howbig := sizeof(ptArray^);
// Clear error bit
q_xError := FALSE;
IF iMessageLen = iCurrIndex THEN
    //Dont do a damn thing
    ;
// Check the remaining length and shift amount summed is not greater than the total array width.
ELSIF iSize < (iMessageLen - iCurrIndex) + iShift THEN
    q_xError := TRUE;
ELSE// MEMMOVE from 1+ the current index to the remaining length by the shift amount
    IF MEMMOVE(srcAddr:=(ptArray + iCurrIndex + 1), destAddr:=(ptArray + iCurrIndex + 1 + iShift), n:=INT_TO_UDINT(iMessageLen + 1 - iCurrIndex)) =0 THEN
        q_xError := TRUE;
    END_IF
END_IF

END_FUNCTION_BLOCK

// ---- POUs/Sensirion/fSHDLCChecksum.TcPOU
FUNCTION fSHDLCChecksum : BYTE
VAR_INPUT
    i_bAdr	:	BYTE;
    i_bCmd	:	BYTE;
    i_bLen	:	BYTE;
    i_pbaTxData	:	POINTER TO BYTE;
END_VAR
VAR
    iIndex	:	INT;
END_VAR

(* Checksum is calc like so
Sum all the bytes within the frame
Take the LSN ie. nibble of the result and invert it
*)

fSHDLCChecksum := i_bAdr + i_bCmd + i_bLen;

IF i_bLen > 0 THEN
FOR iIndex:=0 TO BYTE_TO_INT(i_bLen)DO
    fSHDLCChecksum := fSHDLCChecksum + i_pbaTxData^;
    i_pbaTxData := i_pbaTxData + 1;
END_FOR
END_IF

// Inverting LSN
fSHDLCChecksum := fSHDLCChecksum XOR 16#FF;

END_FUNCTION

// ---- POUs/PCM/FB_PressureControlModule.TcPOU
// Encapsulation of a pressure control module.
// A. Wallace, 2019-10-22
// Support for 2 proportionairs, 4 generic analog inputs (usually a pressure gauge
// and two shimadzu ports.
FUNCTION_BLOCK FB_PressureControlModule
VAR_INPUT
END_VAR
VAR_OUTPUT
END_VAR
VAR_IN_OUT
END_VAR
VAR
    {attribute 'pytmc' := '
        pv: IO
     '}
    stBaseIO : ST_M3DeviceBaseIO;

    stSerial1 : ST_SerialComm;
    stSerial2 : ST_SerialComm;

    fbSerial1 : FB_SerialCommWrapper;
    fbSerial2 : FB_SerialCommWrapper;

    {attribute 'pytmc' := '
        pv: PropAir:01
     '}
    stPropAir1 : ST_Proportionair;
    {attribute 'pytmc' := '
        pv: PropAir:02
     '}
    stPropAir2 : ST_Proportionair;

    PropAir1 : FB_ProportionairRegulator;
    PropAir2 : FB_ProportionairRegulator;
END_VAR

PropAir1(iq_stRegProp:=stPropAir1);
PropAir2(iq_stRegProp:=stPropAir2);

ACTION SerialComm:
fbSerial1(stSerialComm := stSerial1);
fbSerial2(stSerialComm := stSerial2);
END_ACTION

END_FUNCTION_BLOCK

// ---- POUs/Regulators/FB_ProportionairRegulator.TcPOU
FUNCTION_BLOCK FB_ProportionairRegulator
VAR_INPUT
END_VAR
VAR_OUTPUT
END_VAR
VAR_IN_OUT
    iq_stRegProp	:	ST_Proportionair;
END_VAR
VAR

END_VAR

(* A. Wallace 2015-10-7
Proportionair regulator control *)

(* Pressure signal conversion, max pressure out 1000 (I think...) *)
iq_stRegProp.iPressure := REAL_TO_INT(1000 * (MAX(0,INT_TO_REAL(iq_stRegProp.i_iPressRB)) / 32767));

iq_stRegProp.iSetpoint := LIMIT(iq_stRegProp.iLoLimit, iq_stRegProp.iSetpoint, iq_stRegProp.iHiLimit);

iq_stRegProp.q_iPressCt := REAL_TO_INT( (INT_TO_REAL(iq_stRegProp.iSetpoint)/1000)*32767);

END_FUNCTION_BLOCK

// ---- POUs/GasManifold/FB_GasManifold.TcPOU
FUNCTION_BLOCK FB_GasManifold
VAR_INPUT
END_VAR
VAR_OUTPUT
END_VAR
VAR
    {attribute 'pytmc' := '
        pv: IO
     '}
    stBaseIO : ST_M3DeviceBaseIO;


    {attribute 'pytmc' := '
        pv: Valve
     '}
    stValve : ARRAY [1..MANIFOLD_VALVES] OF ST_ManifoldValve;
    fbValve : ARRAY [1..MANIFOLD_VALVES] OF FB_ManiValve;
    idx : int;
END_VAR
VAR CONSTANT
    MANIFOLD_VALVES : INT := 7;
END_VAR

FOR idx := 1 to MANIFOLD_VALVES DO
    stValve[idx].xILK := TRUE; // these valves have no interlock
    fbValve[idx](iq_valve := stValve[idx]);
END_FOR

END_FUNCTION_BLOCK

// ---- POUs/GasManifold/FB_ManiValve.TcPOU
FUNCTION_BLOCK FB_ManiValve
VAR_INPUT
END_VAR
VAR_OUTPUT
END_VAR
VAR_IN_OUT
    iq_valve	:	ST_ManifoldValve;
END_VAR
VAR
END_VAR

(* Basic valve control block *)
IF NOT iq_valve.xILK THEN
    iq_valve.xSW := FALSE;
END_IF

iq_valve.qxDO := NOT (iq_valve.xILK and iq_valve.xSW); // These are normally open valves, qxDO closes the valve

END_FUNCTION_BLOCK

// ---- POUs/Bronkhorst/FB_BronkhorstMFM.TcPOU
FUNCTION_BLOCK FB_BronkhorstMFM
VAR_INPUT
END_VAR
VAR_OUTPUT
END_VAR
VAR
        {attribute 'pytmc' := '
            pv:
         '}
        stMFM	:	ST_BhElFlow;
END_VAR

END_FUNCTION_BLOCK

// ---- POUs/DigitalOutput/FB_SolenoidPair.TcPOU
FUNCTION_BLOCK FB_SolenoidPair
VAR_INPUT
END_VAR
VAR_OUTPUT
END_VAR
VAR_IN_OUT
END_VAR
VAR
    {attribute 'pytmc' := '
        pv: Valve:01:Open
        io: io
     '}
    q_xDO1 AT %Q*	:	BOOL;
    {attribute 'pytmc' := '
        pv: Valve:02:Open
        io: io
     '}
    q_xDO2 AT %Q*	:	BOOL;

    {attribute 'pytmc' := '
        pv: Switch
        io: o
     '}
    i_xEpics AT %I* : BOOL; // open A when False, open B when True

    {attribute 'pytmc' := '
        pv: Debug
        io: o
     '}
    i_xDebug AT %I* : BOOL; // if True, do not set valves according to i_xEpics
END_VAR

(* If debug, set independently. Else, only open one valve according to i_xEpics *)
IF NOT i_xDebug THEN
    q_xDO1 := NOT i_xEpics;
    q_xDO2 := i_xEpics;
END_IF

END_FUNCTION_BLOCK

// ---- POUs/Helpers/FB_EcatDiag.TcPOU
FUNCTION_BLOCK FB_EcatDiag
VAR_INPUT
    i_AMSNetId	:	AMSNETID; //Connect this to an AMSNETID structure as a PLC input. Then link the input to the AMSNETID name in the master info.
    i_xFirstPass	:	BOOL;
END_VAR
VAR_OUTPUT
    q_xAllStatesGood	:	BOOL;
END_VAR
VAR
    sNetId : T_AmsNetId;
    astTermStates : ARRAY[1..256] OF ST_EcSlaveState;

    fbGetAllSlaveStates     : FB_EcGetAllSlaveStates;
    ftReset	: F_TRIG;

    iterator: INT;
END_VAR

//Create the net ID string
sNetID := F_CreateAmsNetId(i_AMSNetId);

//Query the state of all terminals, collect in astTermStates
ftReset(CLK:=fbGetAllSlaveStates.bBusy OR i_xFirstPass);
fbGetAllSlaveStates.bExecute := ftReset.Q;
fbGetAllSlaveStates(sNetId:=sNetId, pStateBuf := ADR(astTermStates), cbBufLen:=SIZEOF(astTermStates));
//Keep checking...

//Cycle through each entry in the array and check if we have anyone not in OP and that the link state is good.
// If so, then set our global IO bad boolean.
IF fbGetAllSlaveStates.nSlaves > 0 THEN
    q_xAllStatesGood := TRUE;
FOR iterator := 1 TO (fbGetAllSlaveStates.nSlaves -1) BY 1
    DO
    IF NOT( (astTermStates[iterator].deviceState = EC_DEVICE_STATE_OP) AND (astTermStates[iterator].linkState = EC_LINK_STATE_OK)) THEN
        q_xAllStatesGood := FALSE;
    END_IF
END_FOR
END_IF

END_FUNCTION_BLOCK

// ---- POUs/p_ALI.TcPOU
PROGRAM p_ALI
VAR
    fbALI_A	:	FB_ALI;
END_VAR

fbALI_A(iq_Injector:=stALI);

END_PROGRAM

// ---- POUs/p_Autosave.TcPOU
PROGRAM p_Autosave
VAR
END_VAR

(* If first pass, copy all persistent variables (which should be intialized to old values) back into the operational variables *)
IF g_xFirstPass THEN

    stRegProp1 := gp_stRegProp1;
    stRegProp2 := gp_stRegProp2;
    stRegProp3 := gp_stRegProp3;
    stRegProp4 := gp_stRegProp4;

ELSE
    gp_stRegProp1 := stRegProp1;
    gp_stRegProp2 := stRegProp2;
    gp_stRegProp3 := stRegProp3;
    gp_stRegProp4 := stRegProp4;

END_IF

END_PROGRAM

// ---- POUs/p_AutoWash.TcPOU
PROGRAM p_AutoWash
VAR



END_VAR

END_PROGRAM

// ---- POUs/p_CoolerShaker.TcPOU
PROGRAM p_CoolerShaker
VAR

afbTECDriver	:	ARRAY[1..3] OF FB_TECDriver;

    index: INT :=1 ;
END_VAR


stTECCtrl[1].sAddress := '01'; //62 is 98 in hex which is default address
stTECCtrl[2].sAddress := '02';
stTECCtrl[3].sAddress := '62';

stTECCtrl[1].diTempSetpoint := 30; //98 in hex which is default address
stTECCtrl[2].diTempSetpoint := 30;
stTECCtrl[3].diTempSetpoint := 30;

afbTECDriver[index](
    i_xExecute:= TRUE,
    i_tTimeOut:= t#1s,
    i_stControl:= stTECCtrl[index],
    iq_stSerialRXBuffer:= SerialRXBuffer_CoolerShakerTEC,
    iq_stSerialTXBuffer:= SerialTXBuffer_CoolerShakerTEC,
    q_stStatus=>stTECStatus[index]);

IF afbTECDriver[index].q_xDone OR
    afbTECDriver[index].q_xError OR
    afbTECDriver[index].q_xTimeout THEN
    (* reset function for next time *)
    afbTECDriver[index](i_xExecute:=FALSE, iq_stSerialRXBuffer:= SerialRXBuffer_CoolerShakerTEC, iq_stSerialTXBuffer:=  SerialTXBuffer_CoolerShakerTEC);

    index := index + 1;
    IF index > 2 THEN index := 1; END_IF

END_IF

END_PROGRAM

// ---- POUs/TEC/FB_TECDriver.TcPOU
FUNCTION_BLOCK FB_TECDriver

VAR_INPUT
    i_xExecute				: BOOL;					(* rising edge execute *)
    i_tTimeOut				: TIME := t#10s;  		(* Maximum wait time for reply *)
    i_stControl				: ST_TECControl;
END_VAR
VAR_OUTPUT
    q_xDone					: BOOL;
    q_xError				: BOOL;
    q_xWarning				: BOOL;					(* set in the event of an unexpected reply *)
    q_xTimeout				: BOOL;
    q_sResult				: STRING(255);
    q_sLastSentString		: ARRAY[1..40] OF STRING;				(* Last String Sent to Serial Device - for debugging *)
    q_sLastReceivedString	: ARRAY[1..40] OF STRING;				(* Last String Received from Serial Device - for debugging *)
    q_stStatus				: ST_TECStatus;
END_VAR
VAR_IN_OUT
    iq_stSerialRXBuffer 	: ComBuffer;
    iq_stSerialTXBuffer 	: ComBuffer;
END_VAR
VAR
    rtExecute				: R_TRIG;
    iStep					: INT;
    sSendData				: STRING;
    fbTECTransaction		: FB_TECTransaction;
    (*fbFormatString			: FB_FormatString;*)
    (*fbSplit					: FB_Split255;*)
    asReplyFields			: ARRAY[1..20] OF T_MaxString;
    wChecksum: WORD;
    rtStartIntegration: R_TRIG;
    rtEndReset: R_TRIG;

    sWorking: STRING;
    strResponseExpected: STRING;
    diWorking	:	DINT;
END_VAR

(* This function block performs serial communication with a TC-36-25 TEC Driver *)

(* rising edge trigger *)
rtExecute(CLK:= i_xExecute);
IF rtExecute.Q  THEN
    q_xDone	:= FALSE;
    q_xError := FALSE;
    q_xWarning := FALSE;
    q_xTimeout := FALSE;
    q_sResult:= '';
    fbTECTransaction( i_xExecute:= FALSE, iq_stSerialRXBuffer:= iq_stSerialRXBuffer, iq_stSerialTXBuffer:= iq_stSerialTXBuffer );  (* reset *)

    iStep := 10;
END_IF

CASE iStep OF
    0: (* idle *)
        ;

    10: (* Get Current Temperature *)
        fbTECTransaction(
            i_xExecute:= TRUE,
            i_sAddress:=i_stControl.sAddress,
            i_sCmd:= '01',
            i_diParameter := 0,
            i_tTimeOut:= i_tTimeOut,
            iq_stSerialRXBuffer:= iq_stSerialRXBuffer,
            iq_stSerialTXBuffer:= iq_stSerialTXBuffer,
            i_CmdFlag :=FALSE);

        IF fbTECTransaction.q_xError THEN
            q_sResult := CONCAT('in Step 10 serial transaction failed with message: ', fbTECTransaction.q_sResult);
            iStep := 9000;
        ELSIF fbTECTransaction.q_xDone THEN
            q_stStatus.sReply := fbTECTransaction.q_sResponseData;
            sWorking :=LEFT(q_stStatus.sReply, 8);
            sWorking := CONCAT('16#', sWorking);
            q_stStatus.diTemp1 := STRING_TO_DINT(sWorking);
            fbTECTransaction( i_xExecute:= FALSE, iq_stSerialRXBuffer:= iq_stSerialRXBuffer, iq_stSerialTXBuffer:= iq_stSerialTXBuffer, i_CmdFlag :=FALSE);  (* reset *)
            iStep := 20;

        END_IF
    20: (* Read setpoint *)
        fbTECTransaction(
            i_xExecute:= TRUE,
            i_sAddress:=i_stControl.sAddress,
            i_sCmd:= '03', // command
            i_diParameter := 0, // always zero for query
            i_tTimeOut:= i_tTimeOut,
            iq_stSerialRXBuffer:= iq_stSerialRXBuffer,
            iq_stSerialTXBuffer:= iq_stSerialTXBuffer,
            i_CmdFlag :=FALSE);

        IF fbTECTransaction.q_xError THEN
            q_sResult := CONCAT('in Step 20 serial transaction failed with message: ', fbTECTransaction.q_sResult);
            iStep := 9000;
        ELSIF fbTECTransaction.q_xDone THEN
            q_stStatus.sReply := fbTECTransaction.q_sResponseData;
            sWorking :=LEFT(q_stStatus.sReply, 8);
            sWorking := CONCAT('16#', sWorking);
            q_stStatus.diSetPoint := STRING_TO_DINT(sWorking);
            fbTECTransaction( i_xExecute:= FALSE, iq_stSerialRXBuffer:= iq_stSerialRXBuffer, iq_stSerialTXBuffer:= iq_stSerialTXBuffer, i_CmdFlag :=FALSE);  (* reset *)
            iStep := 25;
        END_IF

    25: (* Read output ON/OFF *)
        fbTECTransaction(
            i_xExecute:= TRUE,
            i_sAddress:=i_stControl.sAddress,
            i_sCmd:= '46', // command
            i_diParameter := 0, // always zero for query
            i_tTimeOut:= i_tTimeOut,
            iq_stSerialRXBuffer:= iq_stSerialRXBuffer,
            iq_stSerialTXBuffer:= iq_stSerialTXBuffer,
            i_CmdFlag :=FALSE);

        IF fbTECTransaction.q_xError THEN
            q_sResult := CONCAT('in Step 25 serial transaction failed with message: ', fbTECTransaction.q_sResult);
            iStep := 9000;
        ELSIF fbTECTransaction.q_xDone THEN
            q_stStatus.sReply := fbTECTransaction.q_sResponseData;
            sWorking :=LEFT(q_stStatus.sReply, 8);
            sWorking := CONCAT('16#', sWorking);
            diWorking := STRING_TO_DINT(sWorking);
            q_stStatus.xOutputOn := DINT_TO_BOOL(diWorking);
            A_ResetTransaction();
            iStep := 30;
        END_IF

    30: (* Read the alarm status *)
        fbTECTransaction(
            i_xExecute:= TRUE,
            i_sAddress:=i_stControl.sAddress,
            i_sCmd:= '05', // command
            i_diParameter := 0, // always zero for query
            i_tTimeOut:= i_tTimeOut,
            iq_stSerialRXBuffer:= iq_stSerialRXBuffer,
            iq_stSerialTXBuffer:= iq_stSerialTXBuffer,
            i_CmdFlag :=FALSE);

        IF fbTECTransaction.q_xError THEN
            q_sResult := CONCAT('in Step 10 serial transaction failed with message: ', fbTECTransaction.q_sResult);
            iStep := 9000;
        ELSIF fbTECTransaction.q_xDone THEN
            q_stStatus.sReply := fbTECTransaction.q_sResponseData;
            sWorking :=LEFT(q_stStatus.sReply, 8);
            sWorking := CONCAT('16#', sWorking);
            diWorking := STRING_TO_DINT(sWorking);

            //Alarm assignment
            q_stStatus.xHiTemp	:=	diWorking.0;
            q_stStatus.xLoTemp	:=	diWorking.1;
            q_stStatus.xLoTemp	:=	diWorking.2;
            q_stStatus.xOverCurrent	:=	diWorking.3;
            q_stStatus.xOpenInput1	:=	diWorking.4;
            q_stStatus.xOpenInput2	:=	diWorking.5;
            q_stStatus.xDriverLowVoltage	:=	diWorking.6;

            fbTECTransaction( i_xExecute:= FALSE, iq_stSerialRXBuffer:= iq_stSerialRXBuffer, iq_stSerialTXBuffer:= iq_stSerialTXBuffer, i_CmdFlag :=FALSE);  (* reset *)
            iStep := 40;
        END_IF

    40: (* Output Power *)
        fbTECTransaction(
            i_xExecute:= TRUE,
            i_sAddress:=i_stControl.sAddress,
            i_sCmd:= '02', // command
            i_diParameter := 0, // always zero for query
            i_tTimeOut:= i_tTimeOut,
            iq_stSerialRXBuffer:= iq_stSerialRXBuffer,
            iq_stSerialTXBuffer:= iq_stSerialTXBuffer,
            i_CmdFlag :=FALSE);

        IF fbTECTransaction.q_xError THEN
            q_sResult := CONCAT('in Step 10 serial transaction failed with message: ', fbTECTransaction.q_sResult);
            iStep := 9000;
        ELSIF fbTECTransaction.q_xDone THEN
            q_stStatus.sReply := fbTECTransaction.q_sResponseData;
            sWorking :=LEFT(q_stStatus.sReply, 8);
            sWorking := CONCAT('16#', sWorking);
            diWorking := STRING_TO_DINT(sWorking);

            q_stStatus.diPercentOut := (diWorking/511)*100; //in percentage

            fbTECTransaction( i_xExecute:= FALSE, iq_stSerialRXBuffer:= iq_stSerialRXBuffer, iq_stSerialTXBuffer:= iq_stSerialTXBuffer, i_CmdFlag :=FALSE);  (* reset *)
            iStep := 5000;
        END_IF

    5000: (* Change Setpoint *)
        IF q_stStatus.diSetpoint <> i_stControl.diTempSetpoint THEN

            fbTECTransaction(
                i_xExecute:= TRUE,
                i_sAddress:=i_stControl.sAddress,
                i_sCmd:= '1c', // command
                i_diParameter := i_stControl.diTempSetpoint,
                i_tTimeOut:= i_tTimeOut,
                iq_stSerialRXBuffer:= iq_stSerialRXBuffer,
                iq_stSerialTXBuffer:= iq_stSerialTXBuffer,
                i_CmdFlag :=TRUE);
            IF fbTECTransaction.q_xError THEN
                q_sResult := CONCAT('in Step 5000 serial transaction failed with message: ', fbTECTransaction.q_sResult);
                iStep := 9000;
            ELSIF fbTECTransaction.q_xDone THEN
                fbTECTransaction(
                     i_xExecute:= FALSE,
                    iq_stSerialRXBuffer:= iq_stSerialRXBuffer,
                    iq_stSerialTXBuffer:= iq_stSerialTXBuffer,
                    i_CmdFlag:=FALSE );  (* reset *)
                iStep := 5010;
            END_IF
        ELSE
            iStep := 5010;
        END_IF

    5010: (* Output ON/OFF *)
        IF q_stStatus.xOutputOn <> i_stControl.xOutputOn THEN

            fbTECTransaction(
                i_xExecute:= TRUE,
                i_sAddress:=i_stControl.sAddress,
                i_sCmd:= '2d', // command
                i_diParameter := BOOL_TO_DINT(i_stControl.xOutputOn),
                i_tTimeOut:= i_tTimeOut,
                iq_stSerialRXBuffer:= iq_stSerialRXBuffer,
                iq_stSerialTXBuffer:= iq_stSerialTXBuffer,
                i_CmdFlag :=TRUE);
            IF fbTECTransaction.q_xError THEN
                q_sResult := CONCAT('in Step 5010 serial transaction failed with message: ', fbTECTransaction.q_sResult);
                iStep := 9000;
            ELSIF fbTECTransaction.q_xDone THEN
                fbTECTransaction(
                     i_xExecute:= FALSE,
                    iq_stSerialRXBuffer:= iq_stSerialRXBuffer,
                    iq_stSerialTXBuffer:= iq_stSerialTXBuffer,
                    i_CmdFlag:=FALSE );  (* reset *)
                iStep := 8000;
            END_IF
        ELSE
            iStep := 8000;
        END_IF


    8000: (* done *)
        q_xDone := TRUE;
        IF q_sResult = '' THEN
            q_sResult := 'Success';
            q_stStatus.xStatusValid := TRUE;
        END_IF
        IF  i_xExecute = FALSE THEN
            q_xDone:= FALSE;
            iStep := 0;
        END_IF

    9000:
        _A_ClearStatus();
        q_xTimeout := fbTECTransaction.q_xTimeout;
        q_xError := TRUE;
        q_stStatus.xStatusValid := FALSE;


END_CASE

q_sLastSentString := fbTECTransaction.q_sLastSentString;
q_sLastReceivedString := fbTECTransaction.q_sLastReceivedString;

ACTION A_ResetTransaction:
fbTECTransaction( i_xExecute:= FALSE, iq_stSerialRXBuffer:= iq_stSerialRXBuffer, iq_stSerialTXBuffer:= iq_stSerialTXBuffer, i_CmdFlag :=FALSE);  (* reset *)
END_ACTION

ACTION _A_ClearStatus:
q_stStatus.sReply := '';
END_ACTION

END_FUNCTION_BLOCK

// ---- POUs/TEC/FB_TECTransaction.TcPOU
FUNCTION_BLOCK FB_TECTransaction
VAR_INPUT
    i_xExecute				: 	BOOL;				(* Rising edge execute *)
    i_sCmd					: 	STRING(2); 			(* Send Data *)
    i_sAddress				:	STRING(2);
    i_diParameter			:	DINT;
    i_tTimeOut				:	TIME := T#10S;  	(* Maximum wait time for reply *)
    i_CmdFlag: BOOL := FALSE;
END_VAR
VAR_OUTPUT
    q_xDone					: BOOL;
    q_sResponseData			: STRING;
    q_xError				: BOOL;
    q_xTimeout				: BOOL;
    q_sResult				: STRING;
    q_sLastSentString		: ARRAY[1..40] OF STRING;			(* Last String Sent to Serial Device - for debugging *)
    q_sLastReceivedString	: ARRAY[1..40] OF STRING;			(* Last String Received from Serial Device - for debugging *)
END_VAR
VAR_IN_OUT
    iq_stSerialRXBuffer 	: ComBuffer;
    iq_stSerialTXBuffer 	: ComBuffer;
END_VAR
VAR
    rtExecute				: R_TRIG;
    iStep					: INT;
    fbClearComBuffer		: ClearComBuffer;
    fbSendString			: SendString;
    fbReceiveString			: ReceiveString;
    sReceivedString			: STRING;
    tonTimeout				: TON;
    sSendString: STRING;
    iStringTx: INT := 1;
    iStringRx: INT := 1;

    iStringTxRx: INT := 1;
    sTxRxString: ARRAY[1..40] OF STRING;

    fbFormatParamString	:	FB_FormatString;
    fbFormatParamZPadString	:	FB_FormatString;
    fbFormatCSString	:	FB_FormatString;
    sParameter: STRING;
    iIndexChkSum: INT;
    wCsSum: WORD;
    udiParameter: UDINT;

END_VAR

(* This function block performs serial transactions with a TC-36-25 TEC Driver  *)

(* rising edge trigger *)
rtExecute(CLK:= i_xExecute);
IF rtExecute.Q THEN
    q_xDone	:= FALSE;
    q_sResponseData := '';
    q_xError := FALSE;
    q_xTimeout := FALSE;
    q_sResult:= '';
    q_sLastSentString[iStringTx] := '';
    q_sLastReceivedString[iStringRx]:= '';
    iStep := 10;
END_IF

CASE iStep OF
    0:
        ; (* idle *)

    10: (* clear com buffers *)
        fbClearComBuffer(Buffer:= iq_stSerialRXBuffer);
        fbClearComBuffer(Buffer:= iq_stSerialTXBuffer);
        (* Reset receive *)
        fbReceiveString(
            Reset:= TRUE,
            ReceivedString:= sReceivedString,
            RXbuffer:= iq_stSerialRXBuffer );
        (* build the string *)
        sSendString := CONCAT(i_sAddress, i_sCmd); (* adding the address and command/query *)
        IF i_CmdFlag THEN
            (* Convert the parameter into an 8-wide hex string twos complemented*)
            udiParameter := DINT_TO_UDINT(i_diParameter);
            fbFormatParamString(sFormat:= '%x', arg1:=F_UDINT(udiParameter)); // first convert to a string
            fbFormatParamZPadString(sFormat:='%08s', arg1:=F_STRING(fbFormatParamString.sOut));// then zero pad, because FB_Format string does not zero-pad hex strings naturally
            sParameter := fbFormatParamZPadString.sOut;
        ELSE
            sParameter := '00000000'; (* send zeros if we're querying *)
        END_IF
        (* Add parameter *)
        sSendString := CONCAT(sSendString, sParameter);

        (* Compute checksum *)
        A_Checksum();

        (* add stx at start *)
        sSendString := CONCAT('*', sSendString);
        (* append checksum *)
        fbFormatCSString(sFormat := '%02x', arg1:=F_WORD(wCsSum));
        sSendString	:= CONCAT(sSendString, fbFormatCSString.sOut);
         (*adding tail *)
        sSendString := CONCAT(sSendString,'$R'); (* add <cr> *)

        IF fbFormatParamString.bError OR fbFormatCSString.bError THEN
            q_sResult := CONCAT('In step 10 fbFormatString resulted in error: ', UDINT_TO_STRING(fbFormatParamString.nErrId));
            iStep := 9000;
        ELSE
            fbSendString( SendString:= sSendString, TXbuffer:= iq_stSerialTXBuffer );
        END_IF
        q_sLastSentString[iStringTx] := sSendString;
        IF iStringTx = 40 THEN iStringTx := 1; ELSE iStringTx := iStringTx +1; END_IF
        iStep := iStep + 10;

    20: (* Finish sending the String *)
        IF fbSendString.Busy THEN
            fbSendString( SendString:= sSendString, TXbuffer:= iq_stSerialTXBuffer );
        ELSIF fbSendString.Error <> 0 THEN
            q_sResult := CONCAT('In step 20 fbSendString resulted in error: ', INT_TO_STRING(fbSendString.Error));
            iStep := 9000;
        ELSIF NOT fbSendString.Busy THEN
            iStep:=iStep + 10;
        END_IF
        tonTimeout(IN:= FALSE);

    30: (* Get reply *)
        fbReceiveString(
            Prefix:= '*',
            Suffix:= '^',
            Timeout:= i_tTimeOut,
            Reset:= FALSE,
            ReceivedString:= sReceivedString,
            RXbuffer:= iq_stSerialRXBuffer );
        tonTimeout(IN:= TRUE, PT:= i_tTimeOut);
        IF fbReceiveString.Error <> 0 THEN
            q_sResult := CONCAT('In step 30 fbReceiveString resulted in error: ', INT_TO_STRING(fbReceiveString.Error));
            iStep := 9000;
        ELSIF fbReceiveString.RxTimeout OR tonTimeout.Q THEN
            q_sResult := 'Serial device failed to reply within timeout period';
            q_xTimeout := TRUE;
            iStep := 9000;
        ELSIF fbReceiveString.StringReceived THEN
            q_sLastReceivedString[iStringRx] := sReceivedString;
            IF iStringRx = 40 THEN iStringRx := 1; ELSE iStringRx := iStringRx +1; END_IF
            IF LEN(sReceivedString) < 2 THEN
                q_sResult := 'Reply too short.';
                iStep := 9000;
            ELSE
                (* Removing stx and ack *)
                q_sResponseData := LEFT(sReceivedString,LEN(sReceivedString)-1);
                q_sResponseData := RIGHT(q_sResponseData,LEN(q_sResponseData)-1);
                (* Checking for error messages *)
                IF q_sResponseData = 'XXXXXXXXc0' THEN
                        q_sResult := 'Checksum error reported by driver';
                        iStep := 9000;
                END_IF
                q_sResult := 'Success.';
                q_xDone:= TRUE;
                iStep := 100;
            END_IF
        END_IF




    100: (* done *)
        IF  i_xExecute = FALSE THEN
            q_xDone:= FALSE;
            iStep := 0;
        END_IF
        IF NOT i_CmdFlag THEN
            sTxRxString[iStringTxRx]:=CONCAT(CONCAT(q_sLastSentString[iStringTx], ' received '), q_sLastReceivedString[iStringRx]);
        END_IF
        IF iStringTxRx = 40 THEN iStringTxRx := 1; ELSE iStringTxRx := iStringTxRx +1; END_IF

    9000:
        q_xError := TRUE;;




END_CASE

ACTION A_Checksum:
wCsSum := 0;

FOR iIndexChkSum := 0 TO (LEN(sSendString) -1) DO
    wCsSum:= wCsSum + BYTE_TO_WORD(sSendString[iIndexChkSum]);
END_FOR
wCsSum	:= wCsSum MOD 256; (* modulo 256 *)
END_ACTION

END_FUNCTION_BLOCK

// ---- POUs/p_ESTOP.TcPOU
PROGRAM p_ESTOP
VAR
    rtEstop : R_TRIG;
END_VAR

(*
Estop checks for a rising edge on the estop global variable then triggeres the following actions
1. Set selector to position 12, the default resting place
2. Set the water regulator to 0
The sheath regulator is not set to zero at this point because we don't want to ice the jet.
*)

rtEstop(CLK:=g_xEstop);

(* Check for E-Stop *)
IF rtEstop.Q THEN
    stSelector.iVici1ReqPos := 12;
    stSelector.iVici2ReqPos := 12;
    stSelector.iSyncReqPos	:= 12;
END_IF

END_PROGRAM

// ---- POUs/p_Manifold.TcPOU
PROGRAM p_Manifold
VAR
    fbManiValve : FB_ManiValve;
END_VAR

(* Valve 1 *)
stGasMani.stManiVlv1.xILK := stGasMani.xOnline;
fbManiValve(iq_valve:=stGasMani.stManiVlv1);

(* Valve 2 *)
stGasMani.stManiVlv2.xILK := stGasMani.xOnline;
fbManiValve(iq_valve:=stGasMani.stManiVlv2);

(* Valve 3 *)
stGasMani.stManiVlv3.xILK := stGasMani.xOnline;
fbManiValve(iq_valve:=stGasMani.stManiVlv3);

(* Valve 4 *)
stGasMani.stManiVlv4.xILK := stGasMani.xOnline;
fbManiValve(iq_valve:=stGasMani.stManiVlv4);

(* Valve 5 *)
stGasMani.stManiVlv5.xILK := stGasMani.xOnline;
fbManiValve(iq_valve:=stGasMani.stManiVlv5);

(* Valve 6 *)
stGasMani.stManiVlv6.xILK := stGasMani.xOnline;
fbManiValve(iq_valve:=stGasMani.stManiVlv6);

(* Valve 7 *)
stGasMani.stManiVlv7.xILK := stGasMani.xOnline;
fbManiValve(iq_valve:=stGasMani.stManiVlv7);

(* Valve 8 *)
stGasMani.stManiVlv8.xILK := stGasMani.xOnline;
fbManiValve(iq_valve:=stGasMani.stManiVlv8);

END_PROGRAM

// ---- POUs/p_Regulators.TcPOU
PROGRAM p_Regulators
VAR

fbRegProp1	:	FB_ProportionairRegulator;
fbRegProp2	:	FB_ProportionairRegulator;
fbRegProp3	:	FB_ProportionairRegulator;
fbRegProp4	:	FB_ProportionairRegulator;

END_VAR

(* Proportionair regulators *)
fbRegProp1(iq_stRegProp:=stRegProp1);
fbRegProp2(iq_stRegProp:=stRegProp2);
fbRegProp3(iq_stRegProp:=stRegProp3);
fbRegProp4(iq_stRegProp:=stRegProp4);

END_PROGRAM

// ---- POUs/p_Shakers.TcPOU
PROGRAM p_Shakers
VAR
END_VAR

END_PROGRAM

// ---- POUs/p_SoftIO.TcPOU
PROGRAM p_SoftIO
VAR
END_VAR

(* Shakers *)
stSelector.stShaker01.i_xSwitch := iq_stM2SelectorA.i_EP2338_Ch5;
stSelector.stShaker02.i_xSwitch := iq_stM2SelectorA.i_EP2338_Ch6;
stSelector.stShaker03.i_xSwitch := iq_stM2SelectorA.i_EP2338_Ch7;
stSelector.stShaker04.i_xSwitch := iq_stM2SelectorA.i_EP2338_Ch8;

iq_stM2SelectorA.q_EP2338_Ch1	:= stSelector.stShaker01.q_xPwrDO;
iq_stM2SelectorA.q_EP2338_Ch2	:= stSelector.stShaker02.q_xPwrDO;
iq_stM2SelectorA.q_EP2338_Ch3	:= stSelector.stShaker03.q_xPwrDO;
iq_stM2SelectorA.q_EP2338_Ch4	:= stSelector.stShaker04.q_xPwrDO;

stSelector2.stShaker01.i_xSwitch := iq_stM2SelectorB.i_EP2338_Ch5;
stSelector2.stShaker02.i_xSwitch := iq_stM2SelectorB.i_EP2338_Ch6;
stSelector2.stShaker03.i_xSwitch := iq_stM2SelectorB.i_EP2338_Ch7;
stSelector2.stShaker04.i_xSwitch := iq_stM2SelectorB.i_EP2338_Ch8;

iq_stM2SelectorB.q_EP2338_Ch1	:= stSelector2.stShaker01.q_xPwrDO;
iq_stM2SelectorB.q_EP2338_Ch2	:= stSelector2.stShaker02.q_xPwrDO;
iq_stM2SelectorB.q_EP2338_Ch3	:= stSelector2.stShaker03.q_xPwrDO;
iq_stM2SelectorB.q_EP2338_Ch4	:= stSelector2.stShaker04.q_xPwrDO;

stRegProp1.iPressureRaw := iq_stPressCtrlA.i_EP4374_Ch1;
stRegProp2.iPressureRaw := iq_stPressCtrlA.i_EP4374_Ch2;

iq_stPressCtrlA.q_EP4374_Ch3 := stRegProp1.iSetpointRaw;
iq_stPressCtrlA.q_EP4374_Ch4 := stRegProp2.iSetpointRaw;

stRegProp3.iPressureRaw := iq_stPressCtrlB.i_EP4374_Ch1;
stRegProp4.iPressureRaw := iq_stPressCtrlB.i_EP4374_Ch2;

iq_stPressCtrlB.q_EP4374_Ch3 := stRegProp3.iSetpointRaw;
iq_stPressCtrlB.q_EP4374_Ch4 := stRegProp4.iSetpointRaw;

stGasMani.xOnline := NOT iq_stM3GasManifold.i_SyncUnitWC;

iq_stM3GasManifold.q_EP2338_Ch1 := stGasMani.stManiVlv1.qxDO;
iq_stM3GasManifold.q_EP2338_Ch2 := stGasMani.stManiVlv2.qxDO;
iq_stM3GasManifold.q_EP2338_Ch3 := stGasMani.stManiVlv3.qxDO;
iq_stM3GasManifold.q_EP2338_Ch4 := stGasMani.stManiVlv4.qxDO;
iq_stM3GasManifold.q_EP2338_Ch5 := stGasMani.stManiVlv5.qxDO;
iq_stM3GasManifold.q_EP2338_Ch6 := stGasMani.stManiVlv6.qxDO;
iq_stM3GasManifold.q_EP2338_Ch7 := stGasMani.stManiVlv7.qxDO;
iq_stM3GasManifold.q_EP2338_Ch8 := stGasMani.stManiVlv8.qxDO;

stGasMani.stManiVlv1.ixOPN := iq_stM3GasManifold.i_EP2338_Ch1;
stGasMani.stManiVlv2.ixOPN := iq_stM3GasManifold.i_EP2338_Ch2;
stGasMani.stManiVlv3.ixOPN := iq_stM3GasManifold.i_EP2338_Ch3;
stGasMani.stManiVlv4.ixOPN := iq_stM3GasManifold.i_EP2338_Ch4;
stGasMani.stManiVlv5.ixOPN := iq_stM3GasManifold.i_EP2338_Ch5;
stGasMani.stManiVlv6.ixOPN := iq_stM3GasManifold.i_EP2338_Ch6;
stGasMani.stManiVlv7.ixOPN := iq_stM3GasManifold.i_EP2338_Ch7;
stGasMani.stManiVlv8.ixOPN := iq_stM3GasManifold.i_EP2338_Ch8;

END_PROGRAM

// ---- POUs/p_VacGaugeSup.TcPOU
PROGRAM p_VacGaugeSup

VAR



END_VAR

END_PROGRAM

// ---- POUs/Regulators/FB_Regulator.TcPOU
FUNCTION_BLOCK FB_Regulator
VAR_INPUT
    iI: INT;
    lrVelocity	:	LREAL := 360;
END_VAR
VAR_OUTPUT
q_asResult: ARRAY [1..20] OF STRING;
q_xError	:	BOOL;
END_VAR
VAR_IN_OUT
    iq_stRegulator	:	ST_Regulator;
END_VAR
VAR


mcPower	:	MC_Power;
mcSetHome	:	MC_SetPosition;
mcReset	:	MC_Reset;
mcMoveAbsolute : ARRAY[1..2] OF MC_MoveAbsolute;
mcStatus : MC_ReadStatus;

mcHalt	:	MC_Halt;

    iPressDiff: INT;
    iTolerance: INT := 50;
    xMoveOK: BOOL;
    iStep: INT;

    indexResult: INT := 1;

    xInitComplete	:	BOOL := FALSE;

    ftBackToAuto	:	F_TRIG;
    iPercSPOld: UINT;
    imcBlockIndex: INT;
    imcBlockIndexPrev : INT;

    rtEnable : R_TRIG;
END_VAR

(* Regulator Function Block *)
(* Alex Wallace, 2014-10-16 *)
(* Modified in 2.5.3 to remove all pressure SP  based code *)

rtEnable(CLK:=iq_stRegulator.xRegEnab);

(* Regulator Pressure Calculation *)
iq_stRegulator.wInPress := LIMIT(0, F_rPressure(iRawVoltage := iq_stRegulator.i_iRawInPress), 10000);
iq_stRegulator.wOutPress := LIMIT(0, F_rPressure(iRawVoltage := iq_stRegulator.i_iRawOutPress), 10000);


(* Basic regulator interlocking *)


(* Check for regulator enable *)
xMoveOK := iq_stRegulator.xRegEnab;
IF NOT xMoveOK THEN
    (*iq_stRegulator.wPressSP := 0; not preferred *)
    iq_stRegulator.xRegEnab := FALSE;
    (* add motor error here *)
END_IF

IF q_xError THEN
    iStep := 9000;
ELSIF rtEnable.Q THEN
    xInitComplete := FALSE;
    iStep := 10;
ELSIF xInitComplete THEN
    iStep := 3000;
END_IF


CASE iStep OF
    0: iStep := 10;
    10:
    (* Start by initializing the motor axis *)
    mcPower.Enable := TRUE;
    iq_stRegulator.lrUpperLimPos := 2887;
    IF mcPower.Status THEN
        xInitComplete := TRUE;
        q_asResult[indexResult] := 'Motor init success';
        indexResult := indexResult + 1;
        iStep := 3000;
    ELSIF mcPower.Error THEN
        mcPower.Enable := FALSE;
        iStep := 9000;
        q_xError	:=	TRUE;
        q_asResult[indexResult] := CONCAT('Initilizing regulator motor in step 10 failed with error code: ', UDINT_TO_STRING(mcPower.ErrorID));
        indexResult := indexResult +1;
    END_IF

    //Knob controls
    3000:

    IF iq_stRegulator.i_iPercSP <> iPercSPOld  AND xMoveOK THEN
        mcMoveAbsolute[imcBlockIndex].Execute := FALSE;
        imcBlockIndex := imcBlockIndex + 1;
        IF imcBlockIndex >2 THEN imcBlockIndex := 1; END_IF
        mcMoveAbsolute[imcBlockIndex].Position := LIMIT(0, UINT_TO_LREAL(iq_stRegulator.i_iPercSP) * iq_stRegulator.lrUpperLimPos/65535, MAX(iq_stRegulator.lrUpperLimPos,1));
        mcMoveAbsolute[imcBlockIndex].Execute := TRUE;
        iPercSPOld := iq_stRegulator.i_iPercSP;
    ELSIF mcMoveAbsolute[imcBlockIndex].Done or mcMoveAbsolute[imcBlockIndex].CommandAborted or mcMoveAbsolute[imcBlockIndex].Busy or mcMoveAbsolute[imcBlockIndex].Error THEN
        mcMoveAbsolute[imcBlockIndex].Execute := FALSE;
    END_IF

    9000:
    (* Error *)
    mcReset.Execute := iq_stRegulator.xRegEnab;
    IF mcReset.Done THEN
        q_xError := FALSE;
        mcReset.Execute := FALSE;
        iStep:=10;
    END_IF

END_CASE

//Reset the debugging index
IF indexResult > 20 THEN indexResult := 1; END_IF

(* Regulator Percentage Open *)
(* Calculate the regulator percentage open, based on 6.5 turns to fully open *)

iq_stRegulator.wPercentageOpen := LREAL_TO_WORD( (iq_stRegulator.stRegulatorMotor.NcToPlc.ActPos / MAX(iq_stRegulator.lrUpperLimPos,1))*100);

(* Run the mc blocks *)
iq_stRegulator.stRegulatorMotor();
ActPower();

mcSetHome(Execute:=NOT(iq_stRegulator.xRegLoLS) AND iq_stRegulator.stRegulatorMotor.Status.StandStill, Axis:=iq_stRegulator.stRegulatorMotor, Position:=0, Mode:=FALSE);
IF NOT iq_stRegulator.xRegHiLS THEN iq_stRegulator.lrUpperLimPos := iq_stRegulator.stRegulatorMotor.NcToPlc.ActPos; END_IF
mcReset(Axis:=iq_stRegulator.stRegulatorMotor);

FOR iI := 1 TO 2 DO
mcMoveAbsolute[iI](Axis := iq_stRegulator.stRegulatorMotor, Velocity:=iq_stRegulator.lrVelocity, BufferMode:=MC_Aborting);
END_FOR

IF mcMoveAbsolute[1].Error OR mcMoveAbsolute[2].Error THEN
    q_xError	:=	TRUE;
    mcMoveAbsolute[1].Execute := FALSE;
    mcMoveAbsolute[2].Execute := FALSE;
    q_asResult[indexResult] := 'Error occured with motion blocks';
    indexResult := indexResult +1;
ELSIF mcPower.Error THEN
    q_xError := TRUE;
    q_asResult[indexResult] := concat('mcPower block error: ', UDINT_TO_STRING(mcPower.ErrorID));
END_IF

ACTION ActPower:
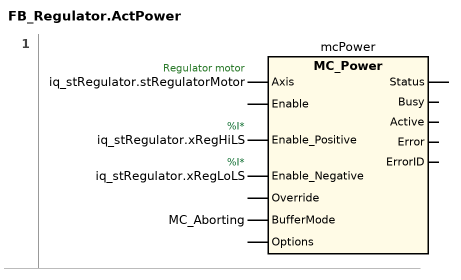
// NETWORK 1
//   iq_stRegulator.stRegulatorMotor: Regulator motor
//   iq_stRegulator.xRegHiLS: AT %I*
//   iq_stRegulator.xRegLoLS: AT %I*
mcPower(
    Axis := iq_stRegulator.stRegulatorMotor,
    Enable_Positive := iq_stRegulator.xRegHiLS,
    Enable_Negative := iq_stRegulator.xRegLoLS,
    BufferMode := MC_Aborting); // MC_Power
END_ACTION

END_FUNCTION_BLOCK

// ---- POUs/Regulators/F_rPressure.TcPOU
FUNCTION F_rPressure : WORD
VAR_INPUT
    iRawVoltage : INT;
END_VAR
VAR
END_VAR

(* Transducer voltage to pressure *)
(* Add formula in here *)
F_rPressure := INT_TO_WORD((iRawVoltage*3000)/32767);

END_FUNCTION

// ---- POUs/p_StatusLights.TcPOU
PROGRAM p_StatusLights
VAR
END_VAR

gxRedLight := xEnableRemoteControl;//Remote control in use
gxGreenLight := NOT (gxRedLight OR gxYellowLight); (* attach system error or something here someday *)

END_PROGRAM
